INTERFACE I_Conveyor

PROPERTY bError : BOOL
GET
END_GET
END_PROPERTY

PROPERTY bMotorRun : BOOL
GET
END_GET
END_PROPERTY

PROPERTY bMotorReverse : BOOL
GET
END_GET
END_PROPERTY

METHOD M_Run
VAR_INPUT
    bForward : BOOL;
END_VAR
END_METHOD

METHOD M_Stop
VAR_INPUT
END_VAR
END_METHOD

METHOD M_Reset
VAR_INPUT
END_VAR
END_METHOD

END_INTERFACE

(* stored: Version 1.1.0.1, ProductVersion 3.1.4024.16
   Itf I_Conveyor: Id {3a4b5c6d-e7f8-9012-abcd-ef1234567890}
   Property bError: Id {4b5c6d7e-f8a9-0123-bcde-f23456789012}
   Get Get: Id {5c6d7e8f-a9b0-1234-cdef-345678901234}
   Property bMotorRun: Id {6d7e8f9a-b0c1-2345-def0-456789012345}
   Get Get: Id {7e8f9a0b-c1d2-3456-ef01-567890123456}
   Property bMotorReverse: Id {8f9a0b1c-d2e3-4567-f012-678901234567}
   Get Get: Id {9a0b1c2d-e3f4-5678-0123-789012345678}
   Method M_Run: Id {0b1c2d3e-f4a5-6789-1234-890123456789}
   Method M_Stop: Id {1c2d3e4f-a5b6-7890-2345-901234567890}
   Method M_Reset: Id {2d3e4f5a-b6c7-8901-3456-012345678901} *)
